% RSLogix 500 project TRAFFIC_LIGHT_6TON_orig.RSS, saved by version 8.30.00.16 %
PROJECT "UNTITLED"    % processor: Bul.1763 MicroLogix 1100 Series A %

PROGRAM FILES
  LAD 2   15 rungs

DATA FILES
  O0 OUTPUT  4 elements
  I1 INPUT  6 elements
  S2 STATUS  66 elements
  B3 BINARY  2 elements
  T4 TIMERS  6 elements
  C5 COUNTER  1 elements
  R6 CONTROL  1 elements
  N7 INTEGER  2 elements
  F8 FLOAT  1 elements

LADDER 2
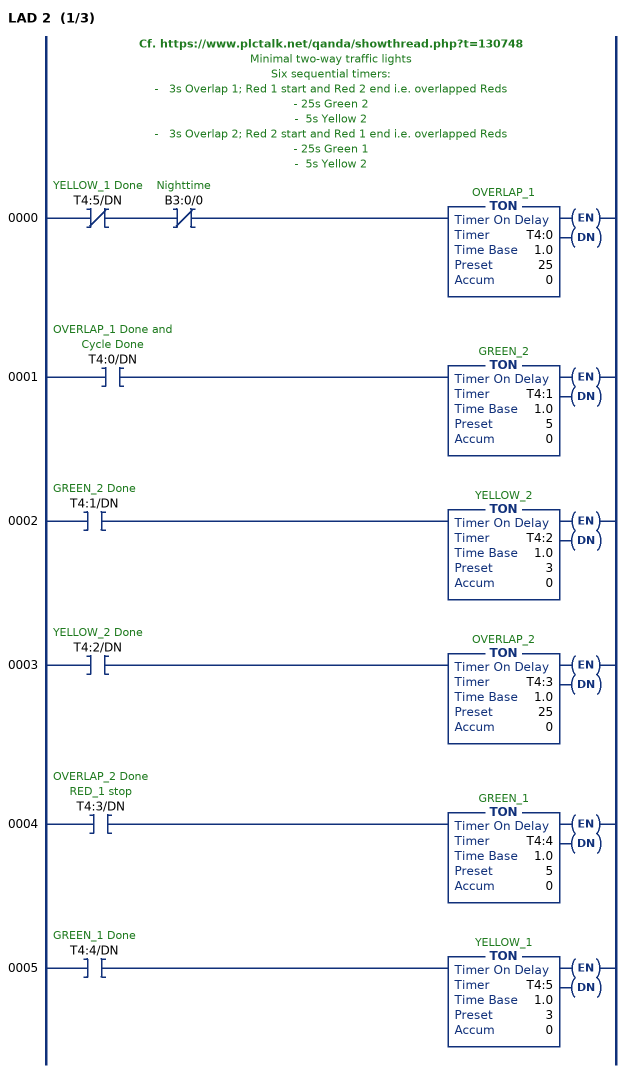
% Rung: 0 %
% TITLE: Cf. https://www.plctalk.net/qanda/showthread.php?t=130748 %
% Minimal two-way traffic lights
% 
% Six sequential timers:
% -   3s Overlap 1; Red 1 start and Red 2 end i.e. overlapped Reds
% - 25s Green 2
% -  5s Yellow 2
% -   3s Overlap 2; Red 2 start and Red 1 end i.e. overlapped Reds
% - 25s Green 1
% -  5s Yellow 2 %
SOR XIO T4:5/DN XIO B3:0/0 TON T4:0 1.0 25 0 EOR
%   T4:5/DN  "YELLOW_1 Done" %
%   B3:0/0  "Nighttime" %
%   T4:0  "OVERLAP_1" %
% Rung: 1 %
SOR XIC T4:0/DN TON T4:1 1.0 5 0 EOR
%   T4:0/DN  "OVERLAP_1 Done and Cycle Done" %
%   T4:1  "GREEN_2" %
% Rung: 2 %
SOR XIC T4:1/DN TON T4:2 1.0 3 0 EOR
%   T4:1/DN  "GREEN_2 Done" %
%   T4:2  "YELLOW_2" %
% Rung: 3 %
SOR XIC T4:2/DN TON T4:3 1.0 25 0 EOR
%   T4:2/DN  "YELLOW_2 Done" %
%   T4:3  "OVERLAP_2" %
% Rung: 4 %
SOR XIC T4:3/DN TON T4:4 1.0 5 0 EOR
%   T4:3/DN  "OVERLAP_2 Done RED_1 stop" %
%   T4:4  "GREEN_1" %
% Rung: 5 %
SOR XIC T4:4/DN TON T4:5 1.0 3 0 EOR
%   T4:4/DN  "GREEN_1 Done" %
%   T4:5  "YELLOW_1" %

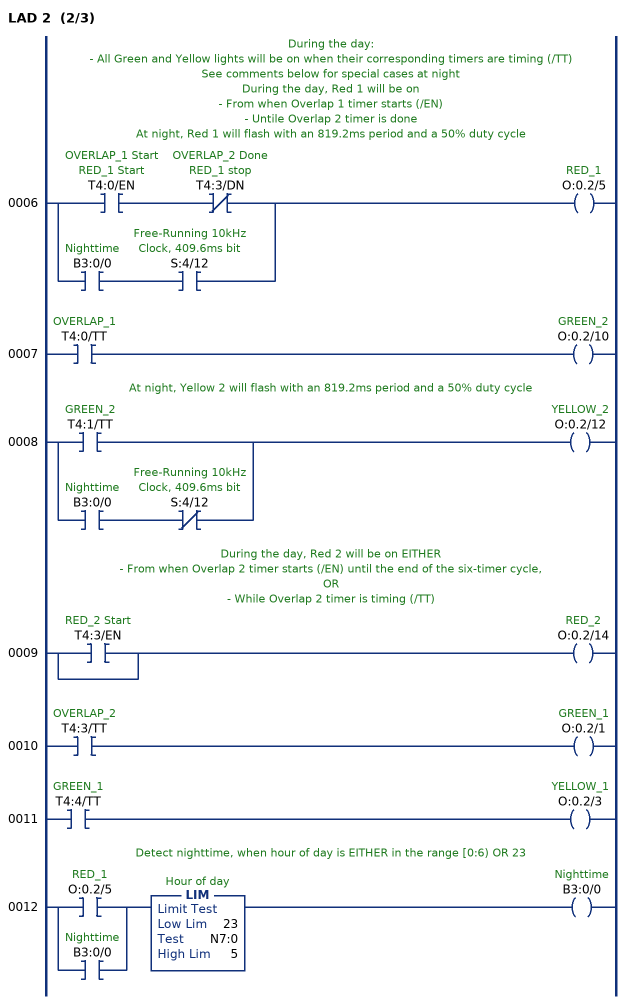
% Rung: 6 %
% During the day:
% - All Green and Yellow lights will be on when their corresponding timers are timing (/TT)
% See comments below for special cases at night
% 
% During the day, Red 1 will be on
% - From when Overlap 1 timer starts (/EN)
% - Untile Overlap 2 timer is done
% At night, Red 1 will flash with an 819.2ms period and a 50% duty cycle %
SOR BST XIC T4:0/EN XIO T4:3/DN NXB XIC B3:0/0 XIC S:4/12 BND OTE O:0.2/5 EOR
%   T4:0/EN  "OVERLAP_1 Start RED_1 Start" %
%   T4:3/DN  "OVERLAP_2 Done RED_1 stop" %
%   B3:0/0  "Nighttime" %
%   S:4/12  "Free-Running 10kHz Clock, 409.6ms bit" %
%   O:0.2/5  "RED_1" %
% Rung: 7 %
SOR XIC T4:0/TT OTE O:0.2/10 EOR
%   T4:0  "OVERLAP_1" %
%   O:0.2/10  "GREEN_2" %
% Rung: 8 %
% At night, Yellow 2 will flash with an 819.2ms period and a 50% duty cycle %
SOR BST XIC T4:1/TT NXB XIC B3:0/0 XIO S:4/12 BND OTE O:0.2/12 EOR
%   T4:1/TT  "GREEN_2" %
%   B3:0/0  "Nighttime" %
%   S:4/12  "Free-Running 10kHz Clock, 409.6ms bit" %
%   O:0.2/12  "YELLOW_2" %
% Rung: 9 %  % edit flag set %
% During the day, Red 2 will be on EITHER
% - From when Overlap 2 timer starts (/EN) until the end of the six-timer cycle,
% OR
% - While Overlap 2 timer is timing (/TT) %
SOR BST XIC T4:3/EN NXB BND OTE O:0.2/14 EOR
%   T4:3/EN  "RED_2 Start" %
%   O:0.2/14  "RED_2" %
% Rung: 10 %
SOR XIC T4:3/TT OTE O:0.2/1 EOR
%   T4:3  "OVERLAP_2" %
%   O:0.2/1  "GREEN_1" %
% Rung: 11 %
SOR XIC T4:4/TT OTE O:0.2/3 EOR
%   T4:4/TT  "GREEN_1" %
%   O:0.2/3  "YELLOW_1" %
% Rung: 12 %
% Detect nighttime, when hour of day is EITHER in the range [0:6) OR 23 %
SOR BST XIC O:0.2/5 NXB XIC B3:0/0 BND LIM 23 N7:0 5 OTE B3:0/0 EOR
%   O:0.2/5  "RED_1" %
%   B3:0/0  "Nighttime" %
%   N7:0  "Hour of day" %

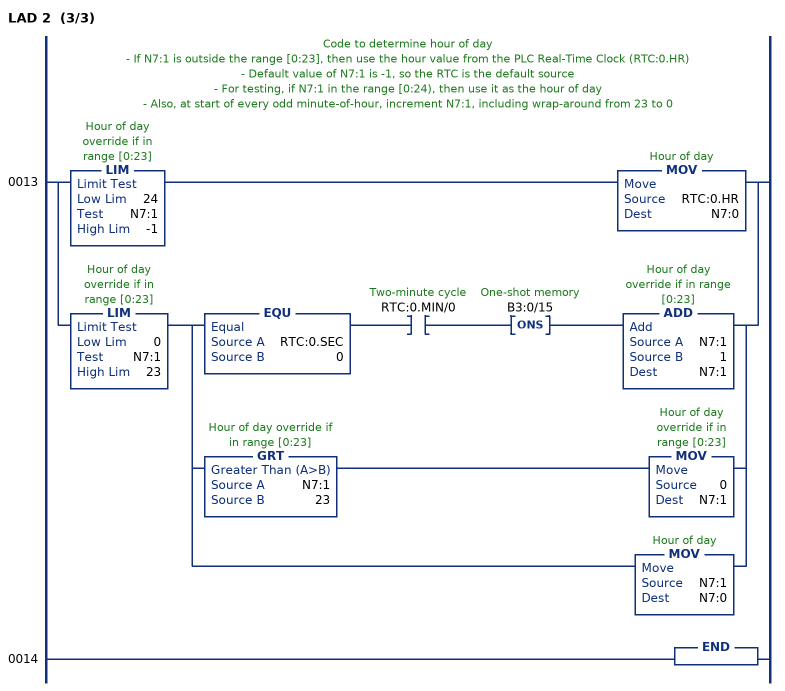
% Rung: 13 %
% Code to determine hour of day
% - If N7:1 is outside the range [0:23], then use the hour value from the PLC Real-Time Clock (RTC:0.HR)
%   - Default value of N7:1 is -1, so the RTC is the default source
% - For testing, if N7:1 in the range [0:24), then use it as the hour of day
%   - Also, at start of every odd minute-of-hour, increment N7:1, including wrap-around from 23 to 0 %
SOR BST LIM 24 N7:1 -1 MOV RTC:0.HR N7:0 NXB LIM 0 N7:1 23 BST EQU RTC:0.SEC 0 XIC RTC:0.MIN/0 ONS B3:0/15 ADD N7:1 1 N7:1 NXB GRT N7:1 23 MOV 0 N7:1 NXB MOV N7:1 N7:0 BND BND EOR
%   N7:1  "Hour of day override if in range [0:23]" %
%   RTC:0.HR  "RTC Hour of day" %
%   N7:0  "Hour of day" %
%   RTC:0.MIN/0  "Two-minute cycle" %
%   B3:0/15  "One-shot memory" %
% Rung: 14 %
SOR END EOR

OTHER DOCUMENTED ADDRESSES
  T4:2/TT  "YELLOW_2"
  T4:5/TT  "YELLOW_1"

DATA TABLE (non-zero values as saved)
DATA T4
% .PRE .ACC %
% T4:0 % 25 0
% T4:1 % 5 0
% T4:2 % 3 0
% T4:3 % 25 0
% T4:4 % 5 0
% T4:5 % 3 0
DATA R6
% .LEN .POS %
% R6:0 % 128 0
DATA N7
% N7:0 % 0 -1
